Fanuc KAREL source: kt00056.KL

-- PROVISIONAL review KL for V940-1; original PC SHA256 a4da270bf5817a24d300796991be40750cbf522658d4d5d88a338917ab6bddd6
-- Incomplete behavior may be omitted. Consult companion uncertainty JSON. Do not deploy.
PROGRAM KT00056
%NOLOCKGROUP
VAR
  OUT : REAL
-- UNRESOLVED_DECL Y1 type=002018
-- UNRESOLVED_DECL H2 type=002017
BEGIN
  -- V9_ZERO_TABLE_METADATA_HINT layout=0001; no indexed target words; source/name/runtime held
  -- UNRESOLVED_PC offsets 5-19; opcodes 2E,22,9D,33,B2
  -- UNRESOLVED_PC offsets 24-38; opcodes 2E,22,9D,33,B4
  -- UNRESOLVED_PC offsets 43-69; opcodes 22,9D,33,B1,22,9D,33,B3,53,64,23
  -- UNRESOLVED_PC offsets 74-78; opcodes 7F
END KT00056
